FUNCTION F_LeakMonitor_LOTAO_2 : FB_LeakMonitor
VAR_INPUT
END_VAR
VAR_OUTPUT
	// Provide stBoundaries output so test functions can reuse the boundaries
	stBoundaries : ST_LeakBoundaries := F_LeakBoundaries();
END_VAR
VAR
	fbLeakMonitor : FB_LeakMonitor;
END_VAR

fbLeakMonitor(
	bLeakDetected := TRUE,
	bAmphosOn := TRUE,
	nLocationResistance := stBoundaries.nLMin1,
	stBound := stBoundaries
);

F_LeakMonitor_LOTAO_2 := fbLeakMonitor;

END_FUNCTION

(* stored: Version 1.1.0.1, ProductVersion 3.1.4024.0
   POU F_LeakMonitor_LOTAO_2: Id {cae9ecbb-6109-42c1-bc29-82d660443624}, SpecialFunc None *)
